FUNCTION_BLOCK FB_AutomaticExtractionStateMachine
VAR_INPUT
	parameters : ST_AutomaticExtractionParameters;
	controlValveFullOpenTime : DINT;
	reactorPressure : DINT;
	pumpPressure : DINT;
	pumpSetpoint : DINT;
END_VAR
VAR_OUTPUT
	controlValveOpeningPercentage : DINT;
	decreasePumpSetpoint : BOOL;
	extractivePumpOn : BOOL;
	co2onOffValveClosed : BOOL;
	fillingActive : BOOL;
	automaticExtractionState : E_AutomaticExtractionState;
	automaticExtractionValues : ST_AutomaticExtractionValues;
END_VAR
VAR
	TON_FillingTimer : TON;
	TON_WaitForValve : TON;
	TON_WaitForPressure : TON;
	TON_KeepExtractivePumpOn : TON;
	startingReactorPRessure : DINT;
	startingPumpSetpoint : DINT;
	startingPumpPressure : DINT;
	endingPumpPressure : DINT;
	TON_FillingPumpWaitTimer : TON;
	
END_VAR

CASE automaticExtractionState OF 
	
	E_AutomaticExtractionState.AUTO_EXTRACTION: // Extraction step
		IF controlValveOpeningPercentage <> parameters.controlValveOpeningValue THEN
			automaticExtractionState := 6;
		END_IF
		fillingActive := FALSE;
		// Start filling timer. When filling timer exceeded, move to filling step
		TON_FillingTimer(
						IN := TRUE,
						PT := TO_TIME(parameters.fillingTime*1000));
		IF TON_FillingTimer.Q THEN
			TON_FillingTimer(IN := FALSE);
			startingPumpSetpoint := pumpSetpoint;// Log setpoint at the moment filling procedure starts
			automaticExtractionState := automaticExtractionState + 1;
		END_IF
		
	E_AutomaticExtractionState.REDUCING_CONTROL_VALVE: // Filling step: Control valve to a small opening
		
		fillingActive := TRUE;
		controlValveOpeningPercentage := 20;
		TON_WaitForValve(
						IN := TRUE,
						PT := TO_TIME(1000));//controlValveFullOpenTime*1000));
		IF TON_WaitForValve.Q THEN
			TON_WaitForValve(IN := FALSE);
			automaticExtractionState := automaticExtractionState + 1;
		END_IF		
	E_AutomaticExtractionState.REDUCING_CO2_PUMP_SETPOINT: // Set pump setpoint to 80 bar
	
		decreasePumpSetpoint := TRUE;
//		TON_WaitForPressure(
//							IN := TRUE,
//							PT := TO_TIME(parameters.pumpSetpointWaitTime*1000));
//		IF TON_WaitForPressure.Q THEN
//			TON_WaitForPressure(IN := FALSE);
//			co2onOffValveClosed := TRUE;  // Close co2 on/off valve
//			automaticExtractionState := automaticExtractionState + 1;
//		END_IF
		IF pumpPressure <= startingPumpSetpoint THEN
			TON_WaitForPressure(IN := FALSE);
			automaticExtractionState := automaticExtractionState + 1;			
		END_IF
		
	E_AutomaticExtractionState.CLOSING_ON_OFF_VALVE:
	
		co2onOffValveClosed := TRUE;  // Close co2 on/off valve
		TON_FillingPumpWaitTimer(IN := TRUE, PT := TO_TIME(parameters.pumpWaitTime*1000));
		IF TON_FillingPumpWaitTimer.Q THEN
			TON_FillingPumpWaitTimer(IN := FALSE);
			startingReactorPressure := reactorPressure;
			startingPumpPressure := pumpPressure;
			automaticExtractionState := automaticExtractionState + 1;		
		END_IF
	
	E_AutomaticExtractionState.FILLING_ACTIVE: //  extractive pump on: stays on for a desired time
	
//		co2onOffValveClosed := TRUE;
		extractivePumpOn := TRUE;
		TON_KeepExtractivePumpOn(
								IN := TRUE,
								PT := TO_TIME(parameters.pumpOnTime*1000));
		IF TON_KeepExtractivePumpOn.Q THEN
			TON_KeepExtractivePumpOn(IN := FALSE);
			endingPumpPressure := pumpPressure;
			automaticExtractionState := automaticExtractionState + 1;
		END_IF
	
	E_AutomaticExtractionState.TURNING_EXTRACTIVE_PUMP_OFF: // Extractive pump turns off after pressure reaches the same as it was b4 turning on
	
		IF (startingReactorPRessure + (startingPumpPressure - endingPumpPressure)) <= reactorPressure THEN
			extractivePumpOn := FALSE;
			automaticExtractionState := automaticExtractionState + 1;
		END_IF
		
	E_AutomaticExtractionState.INCREASING_CO2_PUMP_SETPOINT: // Pressure setpoint back to original (+40bar) and open on/off valve
	
		co2onOffValveClosed := FALSE;
		decreasePumpSetpoint := FALSE;
		automaticExtractionState := automaticExtractionState + 1;
	
	E_AutomaticExtractionState.OPENING_CONTROL_VALVE_TO_SETPOINT: // open control valve to desired value
	
		controlValveOpeningPercentage := parameters.controlValveOpeningValue;
		automaticExtractionState := 0;
		
END_CASE

METHOD getCurrentTimer : BOOL
VAR_INPUT
END_VAR

CASE automaticExtractionState OF 
	
	E_AutomaticExtractionState.AUTO_EXTRACTION: // Extraction step

		automaticExtractionValues.currentTimer := TON_FillingTimer.PT;
		automaticExtractionValues.elapsedTime := TON_FillingTimer.ET;
		automaticExtractionValues.timeVisible := TRUE;
		
	E_AutomaticExtractionState.REDUCING_CONTROL_VALVE: // Filling step: Control valve to a small opening
		
		automaticExtractionValues.currentTimer := TON_WaitForValve.PT;
		automaticExtractionValues.elapsedTime := TON_WaitForValve.ET;
		automaticExtractionValues.timeVisible := TRUE;
	
	E_AutomaticExtractionState.REDUCING_CO2_PUMP_SETPOINT: // Set pump setpoint to 80 bar

		automaticExtractionValues.timeVisible := FALSE;	
		
	E_AutomaticExtractionState.CLOSING_ON_OFF_VALVE:
	
		automaticExtractionValues.currentTimer := TON_FillingPumpWaitTimer.PT;
		automaticExtractionValues.elapsedTime := TON_FillingPumpWaitTimer.ET;
		automaticExtractionValues.timeVisible := TRUE;

	E_AutomaticExtractionState.FILLING_ACTIVE: //  extractive pump on: stays on for a desired time
	
		automaticExtractionValues.currentTimer := TON_KeepExtractivePumpOn.PT;
		automaticExtractionValues.elapsedTime := TON_KeepExtractivePumpOn.ET;
		automaticExtractionValues.timeVisible := TRUE;
	
	E_AutomaticExtractionState.TURNING_EXTRACTIVE_PUMP_OFF: // Extractive pump turns off after pressure reaches the same as it was b4 turning on

		automaticExtractionValues.timeVisible := FALSE;	
		
	E_AutomaticExtractionState.INCREASING_CO2_PUMP_SETPOINT: // Pressure setpoint back to original (+40bar) and open on/off valve

		automaticExtractionValues.timeVisible := FALSE;	
	
	E_AutomaticExtractionState.OPENING_CONTROL_VALVE_TO_SETPOINT: // open control valve to desired value

		automaticExtractionValues.timeVisible := FALSE;	

END_CASE
END_METHOD

METHOD resetState : BOOL
VAR_INPUT
END_VAR

automaticExtractionState := 0;
TON_FillingTimer(IN :=FALSE);
TON_WaitForValve(IN :=FALSE);
TON_WaitForPressure(IN :=FALSE);
TON_KeepExtractivePumpOn(IN :=FALSE);
co2onOffValveClosed := FALSE;
decreasePumpSetpoint := FALSE;
extractivePumpOn := FALSE;
fillingActive := FALSE;
END_METHOD

END_FUNCTION_BLOCK

(* stored: Version 1.1.0.1, ProductVersion 3.1.4024.9
   POU FB_AutomaticExtractionStateMachine: Id {fd3c0490-089c-4717-a34f-489c595512a4}, SpecialFunc None
   Method getCurrentTimer: Id {a3ee8146-ea9a-4d24-ba76-03659dc48839}
   Method resetState: Id {bf1ce1ba-fd70-4c2a-963b-7e4edcae03f9} *)
